TYPE ST_DocumentMemento :
STRUCT
	sContent		: STRING;
END_STRUCT
END_TYPE

(* stored: Version 1.1.0.1
   DUT ST_DocumentMemento: Id {7629035c-dc15-47af-a8b2-9fc25fc82d71} *)
